PROGRAM MAIN
VAR
END_VAR

END_PROGRAM

(* stored: Version 1.1.0.1, ProductVersion 3.1.4024.16
   POU MAIN: Id {df4810ca-f672-4106-8e6a-9f89c96327ca}, SpecialFunc None *)
